{attribute 'GeneratedUsingTerminal: EK1110-0000-0017'}
{attribute addProperty VendorId "#x00000002"}
{attribute addProperty BoxType "EK1110-0000-0017"}
{attribute addProperty Description "EK1110 EtherCAT extension"}
{attribute addProperty Physics "KY"}
{attribute addProperty Id "InfoDataAT %I*InfoData_6F19DB2B2"}
{attribute addProperty CRC "532711307"}
{attribute addProperty Size "2"}
TYPE EK1110_1FC0878B EXTENDS TcoIo.EtcSlaveTerminalBase_947E5A46 :
STRUCT
	{attribute addProperty Name "InfoData"}
	InfoData : TcoIo.InfoData_6F19DB2B;
END_STRUCT
END_TYPE

(* stored: Version 1.2.0.0, ProductVersion 3.1.4024.11
   DUT EK1110_1FC0878B: Id {5b152cd5-c873-4dba-a397-92d5abd671ef} *)
